(* Logix 5000 project; controller Reto3_PID Emulate 5570 rev 30.12; software revision 30.00 *)

TASK Alarma (periodic, rate 10 ms, priority 10, watchdog 500 ms) : Alarma_sensores
TASK Escalizaciones (periodic, rate 10 ms, priority 10, watchdog 500 ms) : Escalizacion_sensores
TASK MainTask (continuous, watchdog 500 ms) : MainProgram

MODULES
   Local : Emulate 5570 (ICP 2, rev 30.12)
END_MODULES

VAR_GLOBAL   (* controller tags *)
   Auto : BOOL;
   Bandera_Flujo : BOOL := 1;
   Bandera_Nivel : BOOL;
   Bandera_start : BOOL := 1;
   Control_Flujo : PID := (CTL := -2146392960, EN := 1, NOZC := 1, INI := 1, OLL := 1, DVNA := 1, PVHA := 1, SP := 16.4, KP := 0.1, KI := 1.0, MAXS := 65.0, MAXO := 100.0, UPD := 0.01, PV := 17.255037, ERR := -0.8550377, MAXI := 10.0, MAXCV := 65.0, MAXTIE := 100.0, DATA[0] := 0.14309536, DATA[1] := -424.73938, DATA[2] := 17.255037, DATA[3] := -0.8550377, DATA[4] := 16.4, DATA[5] := 1.5384616, DATA[6] := 6.5, DATA[7] := 0.16, DATA[8] := 0.1, DATA[9] := 1.0, DATA[11] := 0.1, DATA[12] := 1.0, DATA[15] := 0.65, DATA[16] := 1.0);
   Control_Nivel : PID := (CTL := 1053312, NOZC := 1, OLH := 1, DVPA := 1, PVHA := 1, SP := 151.04639, KP := 1.0, KI := 5.0, KD := 0.1, MAXS := 300.0, SO := 100.0, MAXO := 100.0, UPD := 0.01, PV := 129.98915, ERR := 21.057236, OUT := 100.0, MAXI := 10.0, MAXCV := 300.0, MAXTIE := 100.0, DATA[0] := 96.43439, DATA[1] := -693.2755, DATA[2] := 129.98915, DATA[3] := 21.057236, DATA[4] := 151.04639, DATA[5] := 0.33333334, DATA[6] := 30.0, DATA[7] := 0.16, DATA[8] := 0.5, DATA[9] := 5.0, DATA[11] := 0.5, DATA[12] := 5.0, DATA[15] := 3.0, DATA[16] := 1.0);
   CT_Auto : BOOL;
   CT_Manual : BOOL := 1;
   CT_SelectFlujo : BOOL := 1;
   CT_SelectNivel : BOOL;
   CT_SetPoint : REAL := 2.521485;
   CT_SetPointSCADA : REAL;
   CT_T_Flujo : REAL := 2.6546211;
   CT_T_Nivel : REAL;
   CT_VDescarga : REAL;
   CT_Vllenado : REAL := 6.0;
   Flujo_H : BOOL;
   Flujo_HH : BOOL;
   Flujo_tanque : REAL := 17.255037;
   INT_OUT_0 : DINT := 16;
   INT_OUT_1 : DINT := 17;
   Manual : BOOL := 1;
   Mult_SetPoint : REAL := 756.44556;
   Mult_SetPoint_F : DINT := 164;
   Mult_Tflujo : REAL := 172.55037;
   Mult_Tnivel : REAL;
   Nivel_H : BOOL;
   Nivel_HH : BOOL;
   Nivel_tanque : REAL;
   Set_point : REAL;
   Set_point_Flujo : REAL := 16.4;
   Set_point_Nivel : REAL := 75.644554;
   Start : BOOL;
   Start_HMI : BOOL;
   Stop : BOOL := 1;
   Stop_HMI : BOOL;
   tolerancia : DINT := 1;
   Tolerancia_neg : DINT := 225;
   Tolerancia_pos : DINT := 227;
END_VAR

PROGRAM Alarma_sensores   (* main routine Alarma_rutina *)

ROUTINE Alarma_rutina   (* ladder *)
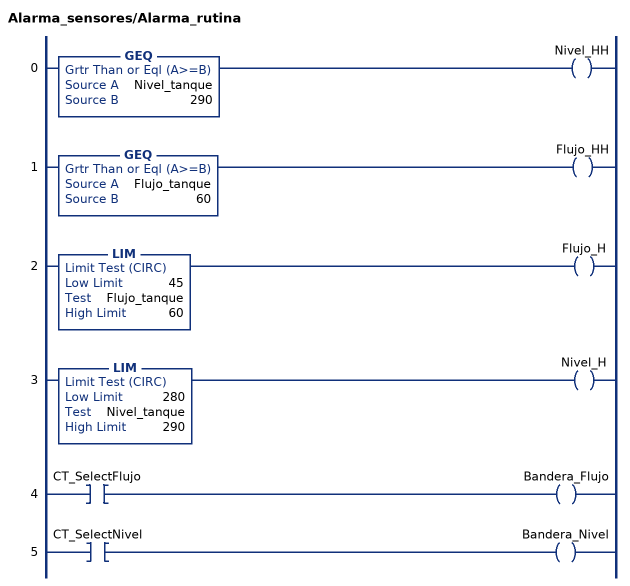
   0: GEQ(Nivel_tanque,290)OTE(Nivel_HH);
   1: GEQ(Flujo_tanque,60)OTE(Flujo_HH);
   2: LIM(45,Flujo_tanque,60)OTE(Flujo_H);
   3: LIM(280,Nivel_tanque,290)OTE(Nivel_H);
   4: XIC(CT_SelectFlujo)OTE(Bandera_Flujo);
   5: XIC(CT_SelectNivel)OTE(Bandera_Nivel);
END_ROUTINE
END_PROGRAM

PROGRAM Escalizacion_sensores   (* main routine Escalizacion_rutina *)

ROUTINE Escalizacion_rutina   (* ladder *)
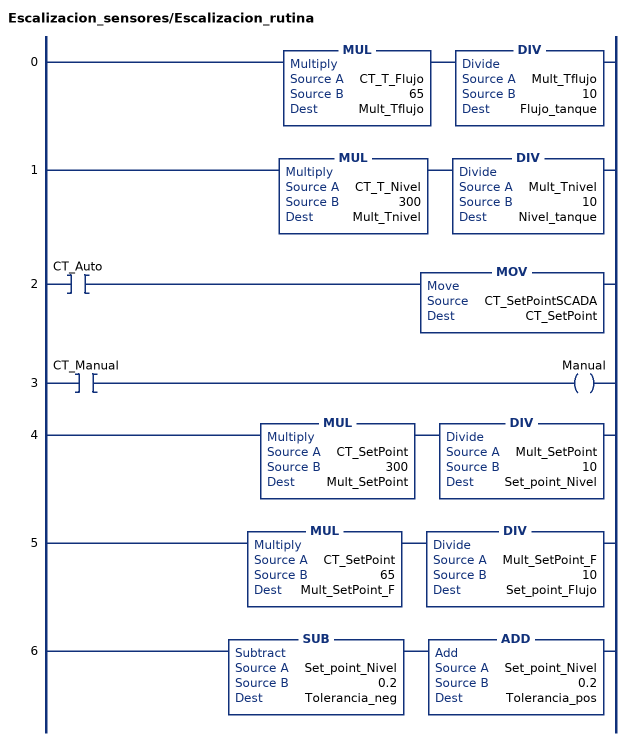
   0: MUL(CT_T_Flujo,65,Mult_Tflujo)DIV(Mult_Tflujo,10,Flujo_tanque);
   1: MUL(CT_T_Nivel,300,Mult_Tnivel)DIV(Mult_Tnivel,10,Nivel_tanque);
   2: XIC(CT_Auto)MOV(CT_SetPointSCADA,CT_SetPoint);
   3: XIC(CT_Manual)OTE(Manual);
   4: MUL(CT_SetPoint,300,Mult_SetPoint)DIV(Mult_SetPoint,10,Set_point_Nivel);
   5: MUL(CT_SetPoint,65,Mult_SetPoint_F)DIV(Mult_SetPoint_F,10,Set_point_Flujo);
   6: SUB(Set_point_Nivel,0.2,Tolerancia_neg)ADD(Set_point_Nivel,0.2,Tolerancia_pos);
END_ROUTINE
END_PROGRAM

PROGRAM MainProgram   (* main routine MainRoutine *)

ROUTINE Flujo   (* ladder *)
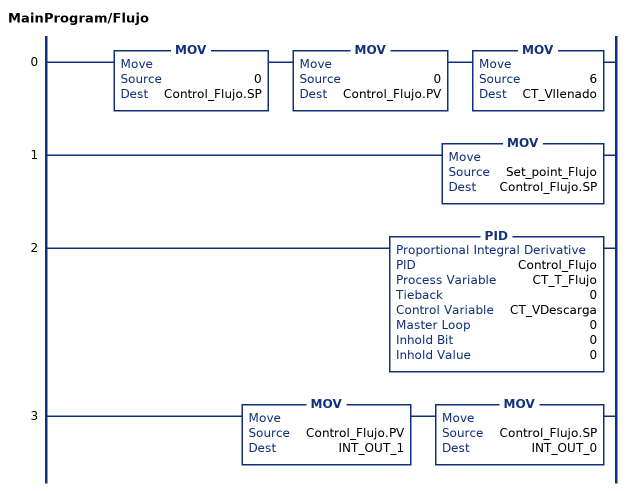
   0: MOV(0,Control_Flujo.SP)MOV(0,Control_Flujo.PV)MOV(6,CT_Vllenado);
   1: MOV(Set_point_Flujo,Control_Flujo.SP);
   2: PID(Control_Flujo,CT_T_Flujo,0,CT_VDescarga,0,0,0);
   3: MOV(Control_Flujo.PV,INT_OUT_1)MOV(Control_Flujo.SP,INT_OUT_0);
END_ROUTINE

ROUTINE MainRoutine   (* ladder *)
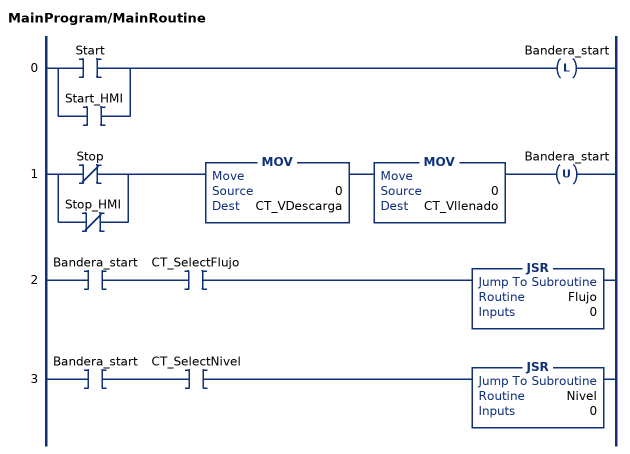
   0: [XIC(Start) ,XIC(Start_HMI) ]OTL(Bandera_start);
   1: [XIO(Stop) ,XIO(Stop_HMI) ]MOV(0,CT_VDescarga)MOV(0,CT_Vllenado)OTU(Bandera_start);
   2: XIC(Bandera_start)XIC(CT_SelectFlujo)JSR(Flujo,0);
   3: XIC(Bandera_start)XIC(CT_SelectNivel)JSR(Nivel,0);
END_ROUTINE

ROUTINE Nivel   (* ladder *)
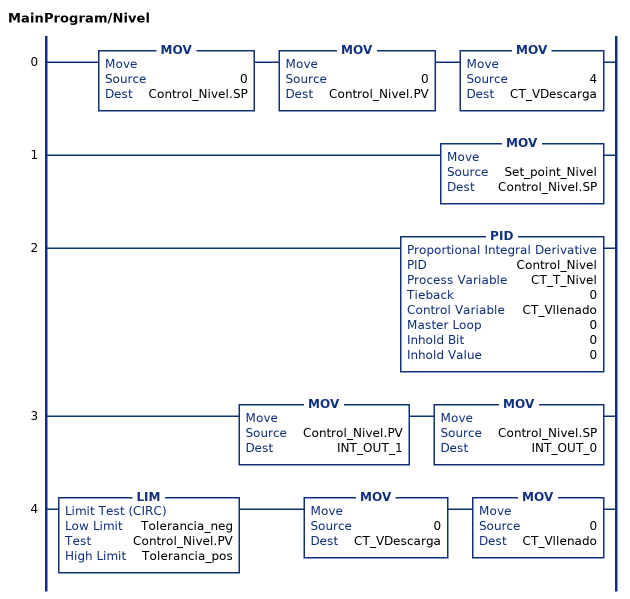
   0: MOV(0,Control_Nivel.SP)MOV(0,Control_Nivel.PV)MOV(4,CT_VDescarga);
   1: MOV(Set_point_Nivel,Control_Nivel.SP);
   2: PID(Control_Nivel,CT_T_Nivel,0,CT_Vllenado,0,0,0);
   3: MOV(Control_Nivel.PV,INT_OUT_1)MOV(Control_Nivel.SP,INT_OUT_0);
   4: LIM(Tolerancia_neg,Control_Nivel.PV,Tolerancia_pos)MOV(0,CT_VDescarga)MOV(0,CT_Vllenado);
END_ROUTINE
END_PROGRAM
